# B&R Automation Studio project DuctLines (part 10)

### Program Logical/E2Buttons (IEC) - This program translates the Coil Line Run, Coil Line Halt And Coil Line Reset Buttons from the touch screen buttons for E2000s.

#### Cyclic.ld
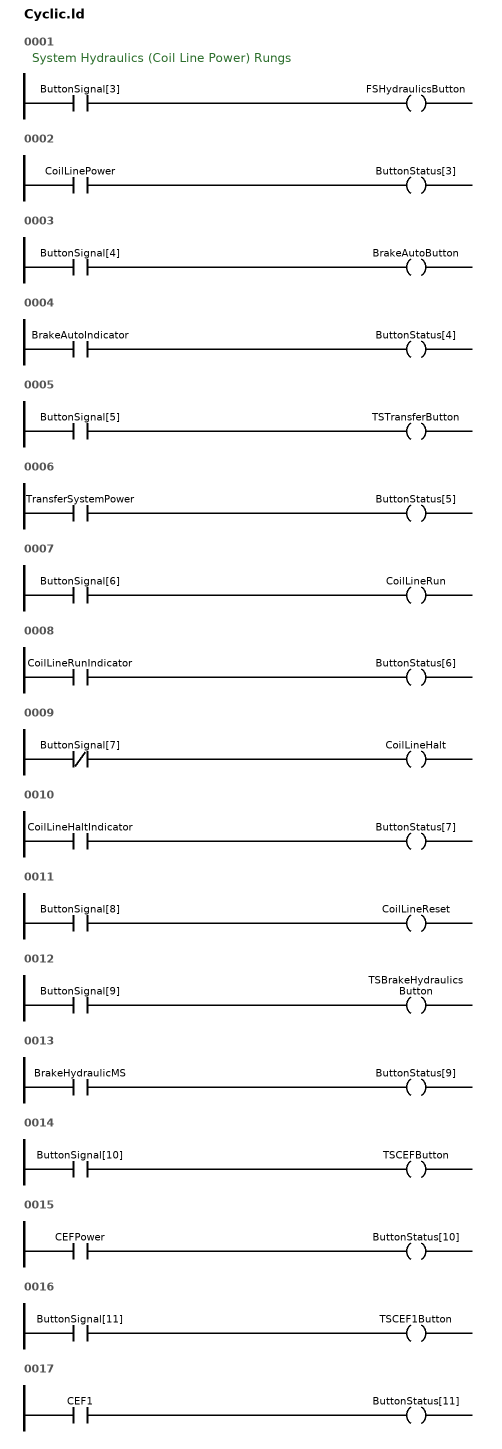
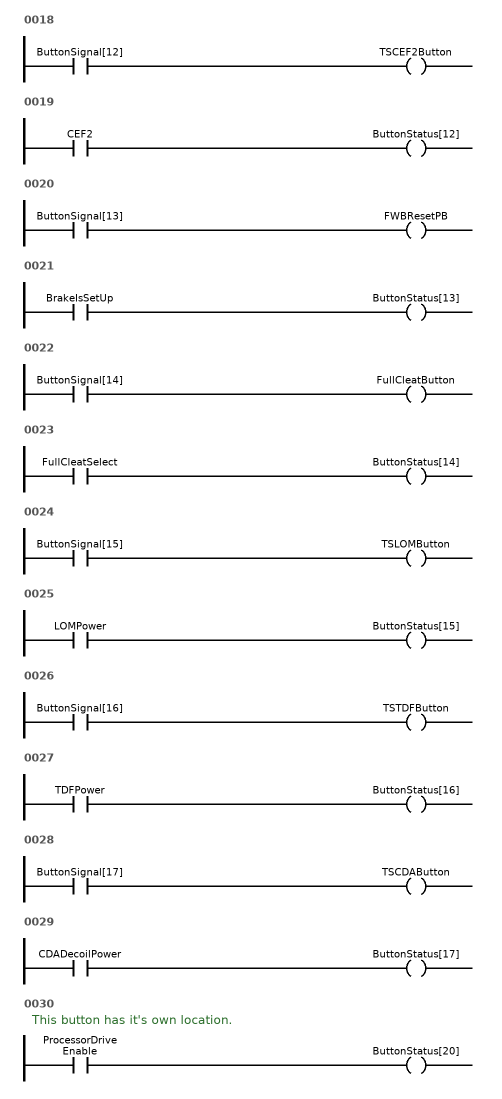
Ladder, written as Structured Text:
```iecst
PROGRAM _CYCLIC
(* Network 1: System Hydraulics (Coil Line Power) Rungs *)
FSHydraulicsButton := ButtonSignal[3];

(* Network 2 *)
ButtonStatus[3] := CoilLinePower;

(* Network 3 *)
BrakeAutoButton := ButtonSignal[4];

(* Network 4 *)
ButtonStatus[4] := BrakeAutoIndicator;

(* Network 5 *)
TSTransferButton := ButtonSignal[5];

(* Network 6 *)
ButtonStatus[5] := TransferSystemPower;

(* Network 7 *)
CoilLineRun := ButtonSignal[6];

(* Network 8 *)
ButtonStatus[6] := CoilLineRunIndicator;

(* Network 9 *)
CoilLineHalt := NOT ButtonSignal[7];

(* Network 10 *)
ButtonStatus[7] := CoilLineHaltIndicator;

(* Network 11 *)
CoilLineReset := ButtonSignal[8];

(* Network 12 *)
TSBrakeHydraulicsButton := ButtonSignal[9];

(* Network 13 *)
ButtonStatus[9] := BrakeHydraulicMS;

(* Network 14 *)
TSCEFButton := ButtonSignal[10];

(* Network 15 *)
ButtonStatus[10] := CEFPower;

(* Network 16 *)
TSCEF1Button := ButtonSignal[11];

(* Network 17 *)
ButtonStatus[11] := CEF1;

(* Network 18 *)
TSCEF2Button := ButtonSignal[12];

(* Network 19 *)
ButtonStatus[12] := CEF2;

(* Network 20 *)
FWBResetPB := ButtonSignal[13];

(* Network 21 *)
ButtonStatus[13] := BrakeIsSetUp;

(* Network 22 *)
FullCleatButton := ButtonSignal[14];

(* Network 23 *)
ButtonStatus[14] := FullCleatSelect;

(* Network 24 *)
TSLOMButton := ButtonSignal[15];

(* Network 25 *)
ButtonStatus[15] := LOMPower;

(* Network 26 *)
TSTDFButton := ButtonSignal[16];

(* Network 27 *)
ButtonStatus[16] := TDFPower;

(* Network 28 *)
TSCDAButton := ButtonSignal[17];

(* Network 29 *)
ButtonStatus[17] := CDADecoilPower;

(* Network 30: This button has it's own location. *)
ButtonStatus[20] := ProcessorDriveEnable;
END_PROGRAM
```

### Program Logical/EFdrSrvDrv (IEC) - Rungs To Control The Electric Servo Drive Option For The Feed Rolls

#### Variables.var
```iecst
VAR
	RollEnableUnlatch : BOOL;
END_VAR
```

#### Cyclic.ld
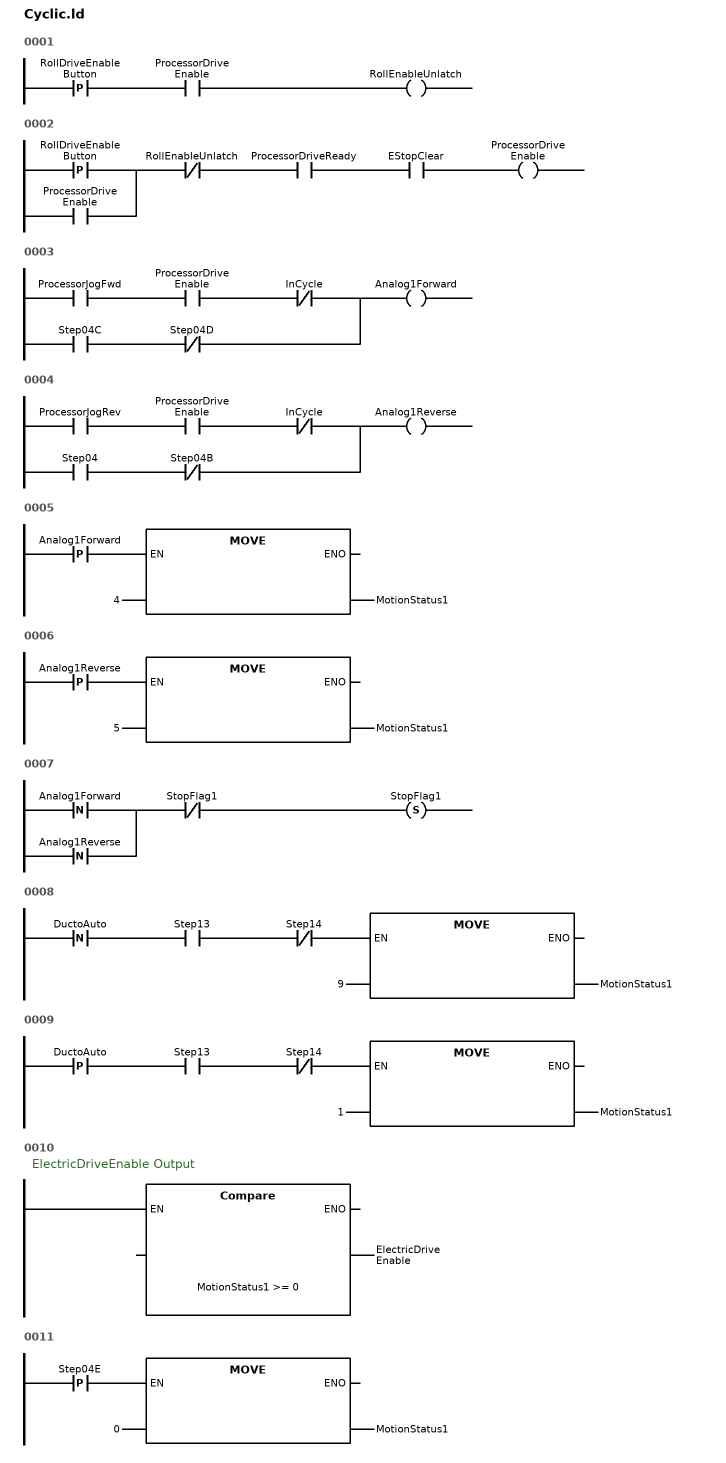
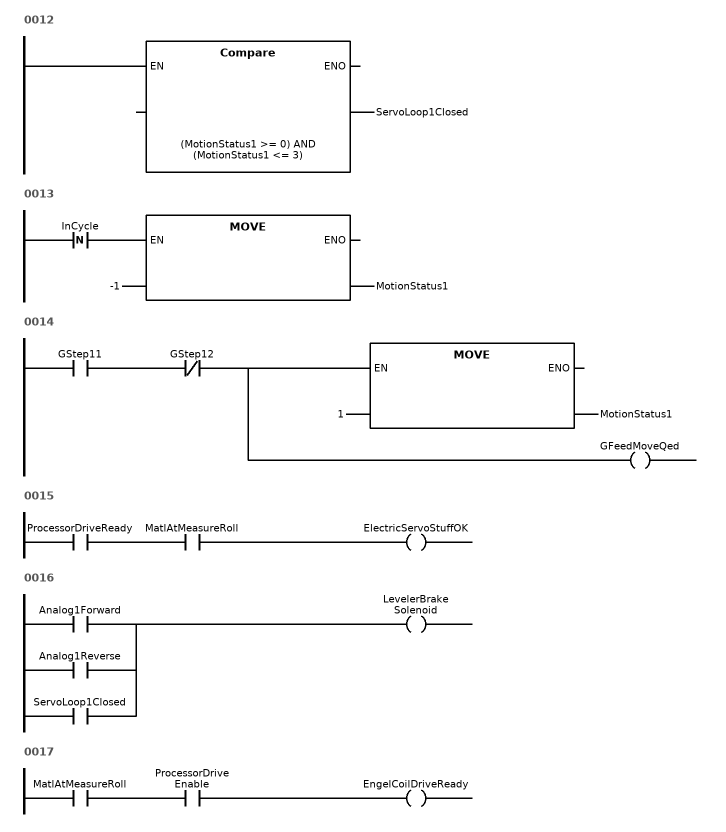
Ladder, written as Structured Text:
```iecst
PROGRAM _CYCLIC
VAR
    _e1 : R_TRIG;
    _e2 : R_TRIG;
    _e3 : R_TRIG;
    _e4 : R_TRIG;
    _e5 : F_TRIG;
    _e6 : F_TRIG;
    _e7 : F_TRIG;
    _e8 : R_TRIG;
    _e9 : R_TRIG;
    _e10 : F_TRIG;
END_VAR
(* Network 1 *)
_e1(CLK := RollDriveEnableButton);
RollEnableUnlatch := _e1.Q AND ProcessorDriveEnable;

(* Network 2 *)
_e2(CLK := RollDriveEnableButton);
ProcessorDriveEnable := (_e2.Q OR ProcessorDriveEnable) AND NOT RollEnableUnlatch AND ProcessorDriveReady AND EStopClear;

(* Network 3 *)
Analog1Forward := (ProcessorJogFwd AND ProcessorDriveEnable AND NOT InCycle) OR (Step04C AND NOT Step04D);

(* Network 4 *)
Analog1Reverse := (ProcessorJogRev AND ProcessorDriveEnable AND NOT InCycle) OR (Step04 AND NOT Step04B);

(* Network 5 *)
_e3(CLK := Analog1Forward);
IF _e3.Q THEN MotionStatus1 := 4; END_IF;

(* Network 6 *)
_e4(CLK := Analog1Reverse);
IF _e4.Q THEN MotionStatus1 := 5; END_IF;

(* Network 7 *)
_e5(CLK := Analog1Forward);
_e6(CLK := Analog1Reverse);
IF (_e5.Q OR _e6.Q) AND NOT StopFlag1 THEN StopFlag1 := TRUE; END_IF;

(* Network 8 *)
_e7(CLK := DuctoAuto);
IF _e7.Q AND Step13 AND NOT Step14 THEN MotionStatus1 := 9; END_IF;

(* Network 9 *)
_e8(CLK := DuctoAuto);
IF _e8.Q AND Step13 AND NOT Step14 THEN MotionStatus1 := 1; END_IF;

(* Network 10: ElectricDriveEnable Output *)
ElectricDriveEnable := MotionStatus1 >= 0;

(* Network 11 *)
_e9(CLK := Step04E);
IF _e9.Q THEN MotionStatus1 := 0; END_IF;

(* Network 12 *)
ServoLoop1Closed := (MotionStatus1 >= 0) AND (MotionStatus1 <= 3);

(* Network 13 *)
_e10(CLK := InCycle);
IF _e10.Q THEN MotionStatus1 := -1; END_IF;

(* Network 14 *)
IF GStep11 AND NOT GStep12 THEN MotionStatus1 := 1; END_IF;
GFeedMoveQed := GStep11 AND NOT GStep12;

(* Network 15 *)
ElectricServoStuffOK := ProcessorDriveReady AND MatlAtMeasureRoll;

(* Network 16 *)
LevelerBrakeSolenoid := Analog1Forward OR Analog1Reverse OR ServoLoop1Closed;

(* Network 17 *)
EngelCoilDriveReady := MatlAtMeasureRoll AND ProcessorDriveEnable;
END_PROGRAM
```

### Program Logical/EFdrHydDrv (IEC) - Rungs to control an Engel processor with the original two speed hydraulic solenoids.

#### Variables.var
```iecst
VAR
	difference : DINT;
	AbsoluteDifference : DINT;
	InTargetWindow : BOOL;
	TON_0 : TON;
	MovingToPosition : BOOL;
	MoveInitiated : BOOL;
	PositionLTTarget : BOOL;
	MoveForward : BOOL;
	PositionGTTarget : BOOL;
	MoveReverse : BOOL;
	InSSWindow : BOOL;
	SettleTimerDone : BOOL;
	TON_1 : TON;
	RevDelay : BOOL;
	TON_2 : TON;
	FwdDelay : BOOL;
	TON_3 : TON;
	SSSDelay : BOOL;
	TON_4 : TON;
	EnableForwardSolenoid : BOOL;
	TP_0 : TP;
	ForwardTP : BOOL;
	TON_5 : TON;
	EnableReverseSolenoid : BOOL;
END_VAR
```

#### Cyclic.ld
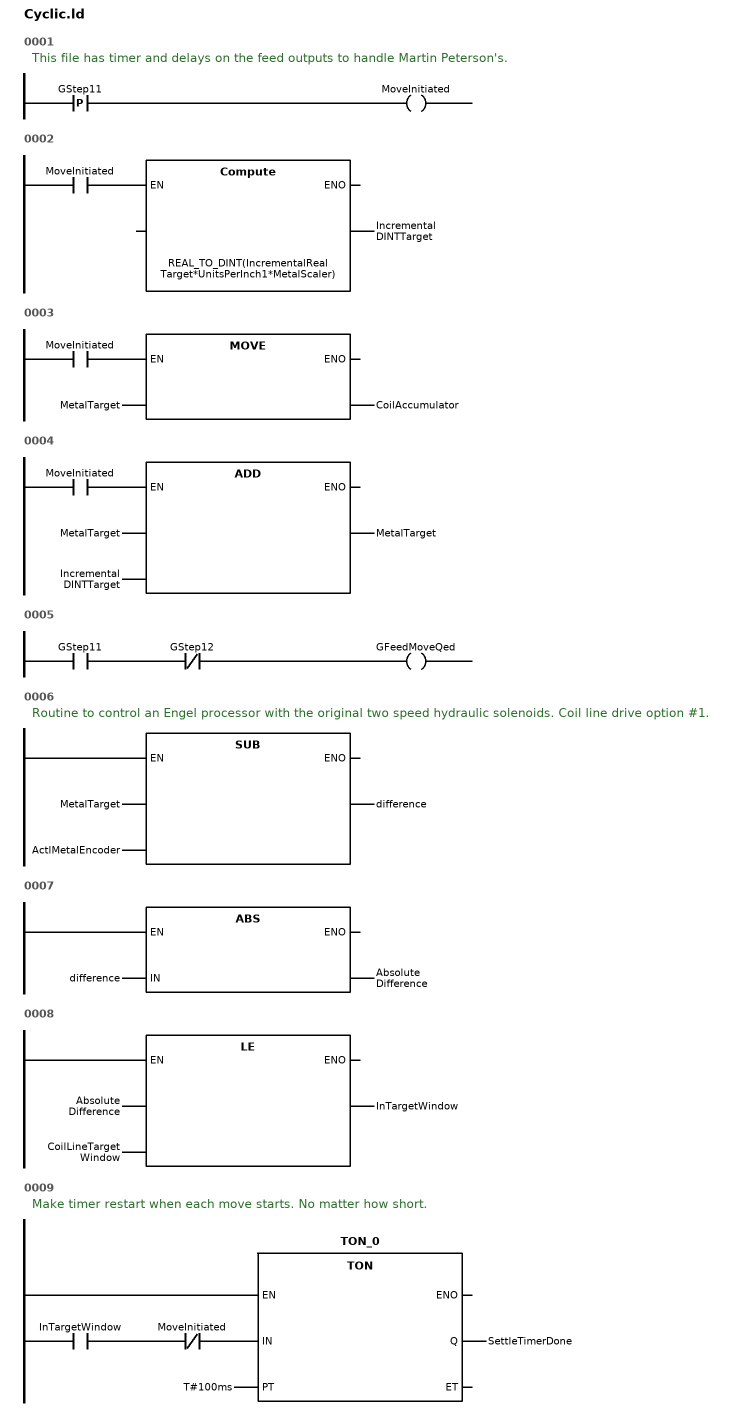
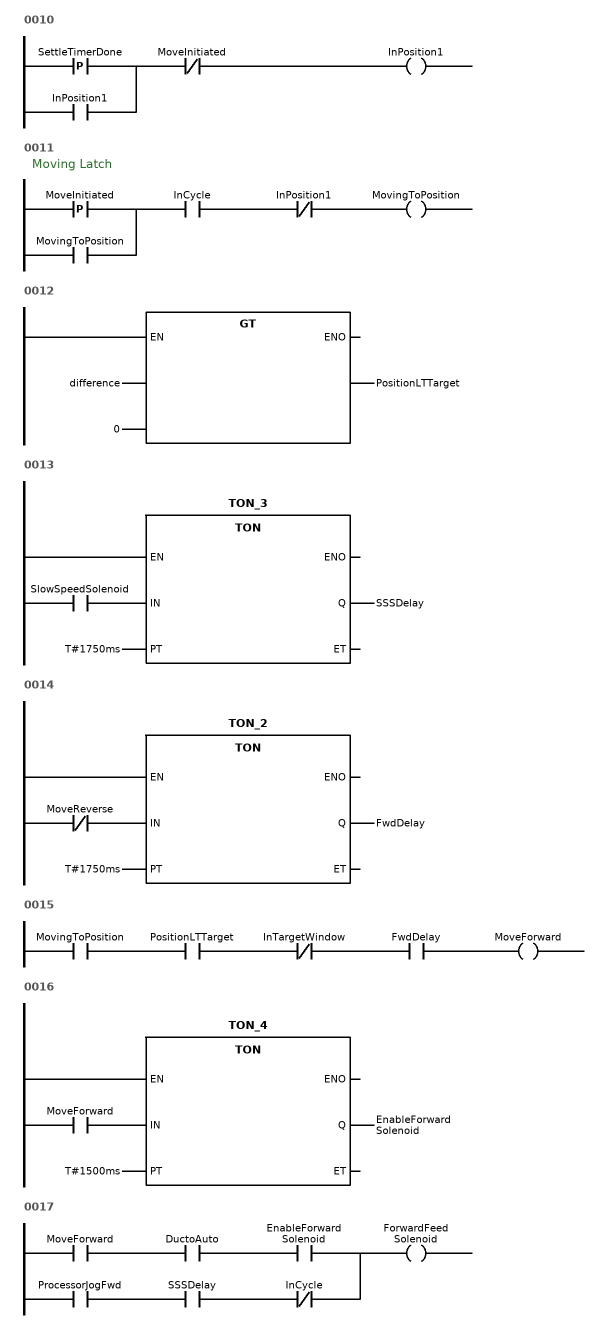
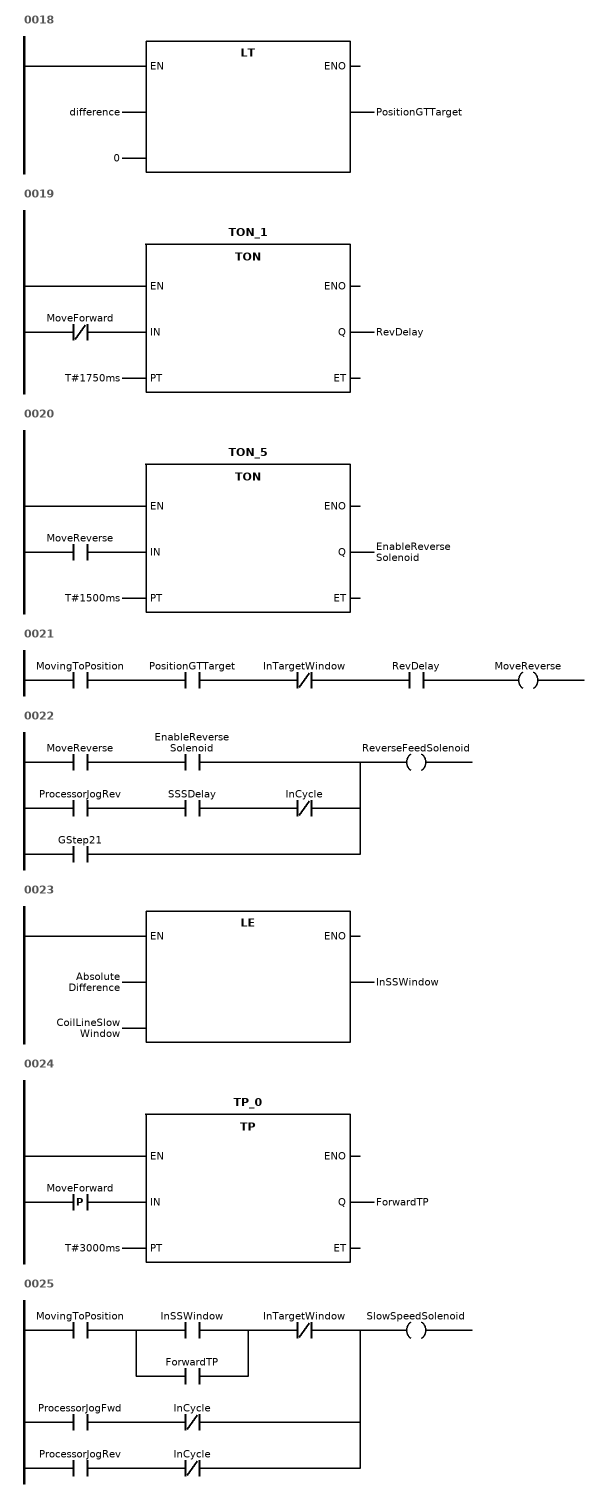
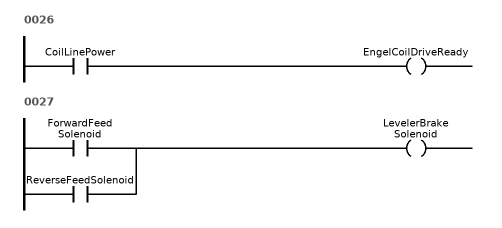
Ladder, written as Structured Text:
```iecst
PROGRAM _CYCLIC
VAR
    _e1 : R_TRIG;
    _e2 : R_TRIG;
    _e3 : R_TRIG;
    _e4 : R_TRIG;
END_VAR
(* Network 1: This file has timer and delays on the feed outputs to handle Martin Peterson's. *)
_e1(CLK := GStep11);
MoveInitiated := _e1.Q;

(* Network 2 *)
IF MoveInitiated THEN
    IncrementalDINTTarget := REAL_TO_DINT(IncrementalRealTarget*UnitsPerInch1*MetalScaler);
END_IF;

(* Network 3 *)
IF MoveInitiated THEN CoilAccumulator := MetalTarget; END_IF;

(* Network 4 *)
IF MoveInitiated THEN MetalTarget := MetalTarget + IncrementalDINTTarget; END_IF;

(* Network 5 *)
GFeedMoveQed := GStep11 AND NOT GStep12;

(* Network 6: Routine to control an Engel processor with the original two speed hydraulic solenoids. Coil line drive option #1. *)
difference := MetalTarget - ActlMetalEncoder;

(* Network 7 *)
AbsoluteDifference := ABS(difference);

(* Network 8 *)
InTargetWindow := AbsoluteDifference <= CoilLineTargetWindow;

(* Network 9: Make timer restart when each move starts. No matter how short. *)
TON_0(IN := InTargetWindow AND NOT MoveInitiated, PT := T#100ms);
SettleTimerDone := TON_0.Q;

(* Network 10 *)
_e2(CLK := SettleTimerDone);
InPosition1 := (_e2.Q OR InPosition1) AND NOT MoveInitiated;

(* Network 11: Moving Latch *)
_e3(CLK := MoveInitiated);
MovingToPosition := (_e3.Q OR MovingToPosition) AND InCycle AND NOT InPosition1;

(* Network 12 *)
PositionLTTarget := difference > 0;

(* Network 13 *)
TON_3(IN := SlowSpeedSolenoid, PT := T#1750ms);
SSSDelay := TON_3.Q;

(* Network 14 *)
TON_2(IN := NOT MoveReverse, PT := T#1750ms);
FwdDelay := TON_2.Q;

(* Network 15 *)
MoveForward := MovingToPosition AND PositionLTTarget AND NOT InTargetWindow AND FwdDelay;

(* Network 16 *)
TON_4(IN := MoveForward, PT := T#1500ms);
EnableForwardSolenoid := TON_4.Q;

(* Network 17 *)
ForwardFeedSolenoid := (MoveForward AND DuctoAuto AND EnableForwardSolenoid) OR (ProcessorJogFwd AND SSSDelay AND NOT InCycle);

(* Network 18 *)
PositionGTTarget := difference < 0;

(* Network 19 *)
TON_1(IN := NOT MoveForward, PT := T#1750ms);
RevDelay := TON_1.Q;

(* Network 20 *)
TON_5(IN := MoveReverse, PT := T#1500ms);
EnableReverseSolenoid := TON_5.Q;

(* Network 21 *)
MoveReverse := MovingToPosition AND PositionGTTarget AND NOT InTargetWindow AND RevDelay;

(* Network 22 *)
ReverseFeedSolenoid := (MoveReverse AND EnableReverseSolenoid) OR (ProcessorJogRev AND SSSDelay AND NOT InCycle) OR GStep21;

(* Network 23 *)
InSSWindow := AbsoluteDifference <= CoilLineSlowWindow;

(* Network 24 *)
_e4(CLK := MoveForward);
TP_0(IN := _e4.Q, PT := T#3000ms);
ForwardTP := TP_0.Q;

(* Network 25 *)
SlowSpeedSolenoid := (MovingToPosition AND (InSSWindow OR ForwardTP) AND NOT InTargetWindow) OR (ProcessorJogFwd AND NOT InCycle) OR (ProcessorJogRev AND NOT InCycle);

(* Network 26 *)
EngelCoilDriveReady := CoilLinePower;

(* Network 27 *)
LevelerBrakeSolenoid := ForwardFeedSolenoid OR ReverseFeedSolenoid;
END_PROGRAM
```

### Program Logical/E2Transfer (IEC) - Controls the E2000 Transfer System

#### Variables.var
```iecst
VAR
	TSPUnlatch : BOOL;
	TSSystemTripPulse : BOOL;
	TP_0 : TP;
	TP_1 : TP;
	TP_2 : TP;
	Lift3DownPulse : BOOL;
	TON_0 : TON;
END_VAR
```

#### Cyclic.ld
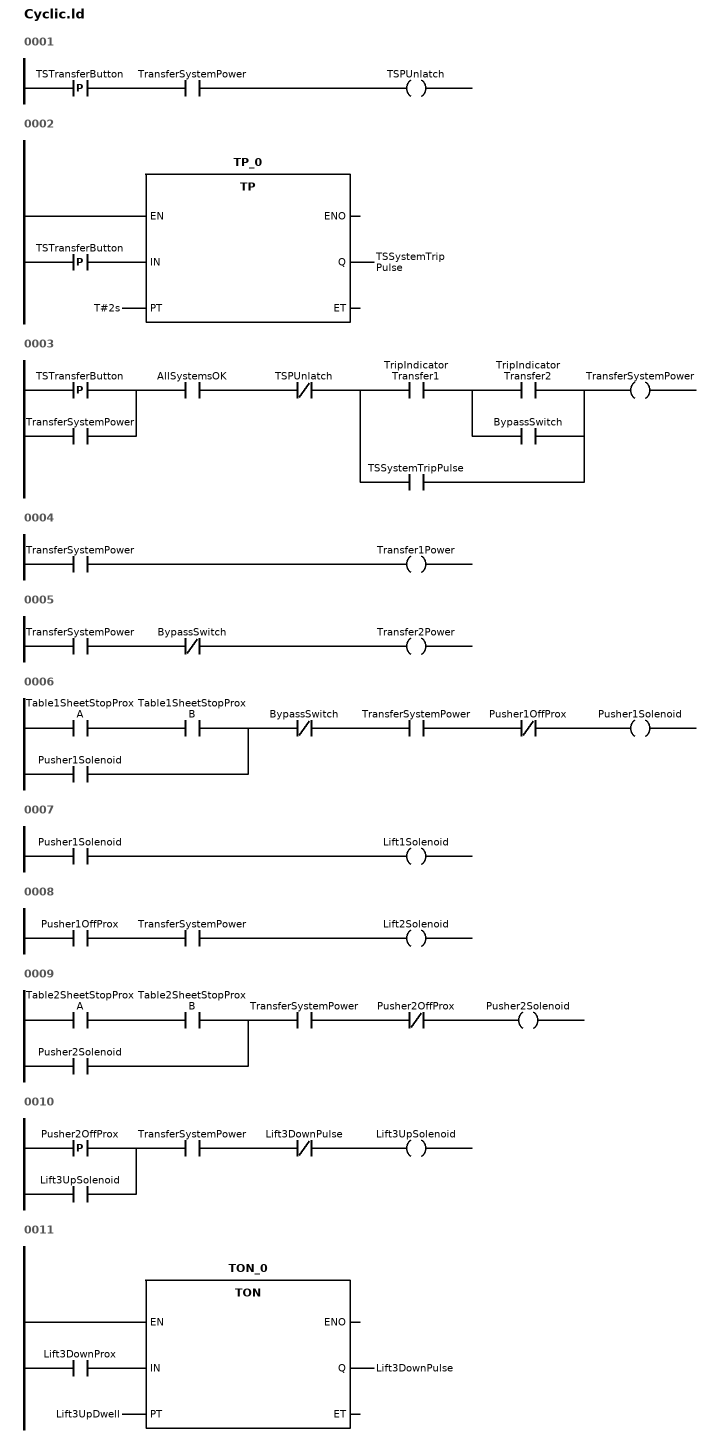
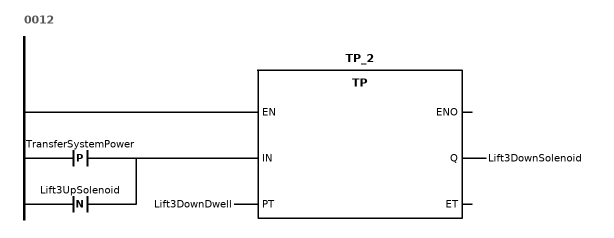
Ladder, written as Structured Text:
```iecst
PROGRAM _CYCLIC
VAR
    _e1 : R_TRIG;
    _e2 : R_TRIG;
    _e3 : R_TRIG;
    _p4 : BOOL;
    _e5 : R_TRIG;
    _e6 : R_TRIG;
    _e7 : F_TRIG;
END_VAR
(* Network 1 *)
_e1(CLK := TSTransferButton);
TSPUnlatch := _e1.Q AND TransferSystemPower;

(* Network 2 *)
_e2(CLK := TSTransferButton);
TP_0(IN := _e2.Q, PT := T#2s);
TSSystemTripPulse := TP_0.Q;

(* Network 3 *)
_e3(CLK := TSTransferButton);
_p4 := (_e3.Q OR TransferSystemPower) AND AllSystemsOK AND NOT TSPUnlatch;
TransferSystemPower := _p4 AND ((TripIndicatorTransfer1 AND (TripIndicatorTransfer2 OR BypassSwitch)) OR TSSystemTripPulse);

(* Network 4 *)
Transfer1Power := TransferSystemPower;

(* Network 5 *)
Transfer2Power := TransferSystemPower AND NOT BypassSwitch;

(* Network 6 *)
Pusher1Solenoid := ((Table1SheetStopProxA AND Table1SheetStopProxB) OR Pusher1Solenoid) AND NOT BypassSwitch AND TransferSystemPower AND NOT Pusher1OffProx;

(* Network 7 *)
Lift1Solenoid := Pusher1Solenoid;

(* Network 8 *)
Lift2Solenoid := Pusher1OffProx AND TransferSystemPower;

(* Network 9 *)
Pusher2Solenoid := ((Table2SheetStopProxA AND Table2SheetStopProxB) OR Pusher2Solenoid) AND TransferSystemPower AND NOT Pusher2OffProx;

(* Network 10 *)
_e5(CLK := Pusher2OffProx);
Lift3UpSolenoid := (_e5.Q OR Lift3UpSolenoid) AND TransferSystemPower AND NOT Lift3DownPulse;

(* Network 11 *)
TON_0(IN := Lift3DownProx, PT := Lift3UpDwell);
Lift3DownPulse := TON_0.Q;

(* Network 12 *)
_e6(CLK := TransferSystemPower);
_e7(CLK := Lift3UpSolenoid);
TP_2(IN := _e6.Q OR _e7.Q, PT := Lift3DownDwell);
Lift3DownSolenoid := TP_2.Q;
END_PROGRAM
```

### Program Logical/EMotionControl (IEC)

#### Variables.var
```iecst
VAR
	AbsoluteDifference : DINT;
	Counter1 : INT;
	DACBalance1 : INT;
	difference : DINT;
	Hold1 : INT;
	Ratio1 : INT;
END_VAR
```

#### Cyclic.st
```iecst
PROGRAM _CYCLIC
	difference := MetalTarget - ActlMetalEncoder;
	AbsoluteDifference := ABS(difference);
	CASE MotionStatus1 OF
		(*Hold Position*)
		0:
			IF NOT InPosition1 THEN
				IF AbsoluteDifference <= MetalTolerance THEN
					TargetCount1 := TargetCount1 + UpdateRate1;
					IF TargetCount1 >= SettleTime1 THEN
						InPosition1 := TRUE;
					END_IF;
				END_IF;
			END_IF;

			(*Ratio1 := DINT_TO_INT(difference + (difference / 1));*)
			Ratio1 := DINT_TO_INT(difference * 15);
			IF Counter1 > 0 THEN
				Counter1 := Counter1 - UpdateRate1;
			ELSE
				Counter1 := 500;
				IF Hold1 <> Ratio1 THEN
					Hold1 := Ratio1;
				ELSE
					DACBalance1 := ActualDAC1;
				END_IF;
			END_IF;

	    	TargetDAC1 := Ratio1 + DACBalance1;
			ActualDAC1 := TargetDAC1;
		(*	IF TargetDAC1 >= ActualDAC1 THEN
				IF TargetDAC1 - ActualDAC1 > (10 * UpdateRate1) THEN
					ActualDAC1 := ActualDAC1 + (10 * UpdateRate1);
				ELSE
					ActualDAC1 := TargetDAC1;
				END_IF;
			ELSE
				IF ActualDAC1 - TargetDAC1 > (10 * UpdateRate1) THEN
					ActualDAC1 := ActualDAC1 - (10 * UpdateRate1);
				ELSE
					ActualDAC1 := TargetDAC1;
				END_IF;
			END_IF;*)

			IF ActualDAC1 > TopDAC1 THEN
				ActualDAC1 := TopDAC1;
			END_IF;
			IF ActualDAC1 < -TopDAC1 THEN
				ActualDAC1 := -TopDAC1;
			END_IF

		(*Initialize Move*)
		1:
			CoilAccumulator := MetalTarget; (*Update Accumulator to last target*)
			(*IncrementalRealTarget is the amount required to move determined elsewhere*)
			IncrementalDINTTarget := REAL_TO_DINT(IncrementalRealTarget * UnitsPerInch1 * MetalScaler);
			MetalTarget := MetalTarget + IncrementalDINTTarget;
			DACAdd1 := INT_TO_REAL(MaxDAC) / AccelRampReal;
			TopDAC1 := DINT_TO_INT((INT_TO_DINT(MaxDAC) * RunSpeed1) / 100);
			IF RunSpeed1 = 100 THEN
				TopDAC1 := TopDAC1 - REAL_TO_INT(DACAdd1);
			END_IF;
			ActualSpeed1 := ((MaxSpeed1 / 5.0) * DINT_TO_REAL(RunSpeed1)) / 100.0; (*Real Inches Per Second*)
			AverageSpeed1 := ActualSpeed1 / 2.0;
			DecelTime1 := (DecelRampReal / 1000.0) * (DINT_TO_REAL(RunSpeed1) / 100);
			DecelDistance1 := REAL_TO_DINT(((AverageSpeed1 * DecelTime1 ) * MetalScaler) * UnitsPerInch1);
			MaxCountsPerSecond := (MaxSpeed1 / 5.0) * UnitsPerInch1;
			SRM1 := MaxDACSquared / ((MaxCountsPerSecond * (DecelRampReal / 1000.0)) / 2.0);
			(*SRM1 := MaxDACSquared / ((MaxCountsPerSecond * (DecelRampReal / 1000.0)));*)
			(*IF DecelDistance1 > IncrementalDINTTarget THEN 2-26-19 *)
			IF DecelDistance1 > (IncrementalDINTTarget / 2) THEN
				DecelDistance1 := IncrementalDINTTarget / 2;
				TopDAC1 := REAL_TO_INT(SQRT((DINT_TO_REAL(DecelDistance1) / MetalScaler) * SRM1));
				IF TopDAC1 < 3276 THEN
					TopDAC1 := 3276;
				END_IF;
			END_IF;
			InPosition1 := FALSE;
			FirstTarget1 := FALSE;
			StopWatch1 := 0.0;
			MotionStatus1 := 2;
		(*Ramp Up To Speed*)
		2:
			IF DecelDistance1 < difference THEN
				IF ActualDAC1 < TopDAC1 THEN (*Accelerate*)
					StopWatch1 := StopWatch1 + INT_TO_REAL(UpdateRate1);
					ActualDAC1 := REAL_TO_INT(StopWatch1 * DACAdd1);
				ELSE  (*Constant Speed*)
					ActualDAC1 := TopDAC1;
				END_IF;
			ELSE (*Switch To Decel MotionState*)
				DecelCounter := 25;
				LastPosition1 := ActlMetalEncoder;
				TargetCount1 := 0;
				FirstTarget1 := FALSE;
				MotionStatus1 := 3;
			END_IF;
		3:
			(*Stall Detection*)
			DecelCounter := DecelCounter - UpdateRate1;
			IF DecelCounter <= 0 THEN
				DecelCounter := 200;
				IF LastPosition1 = ActlMetalEncoder THEN
					DACBalance1 := ActualDAC1;
					Counter1 := 0;
					TopDAC1 := MaxDAC / 4;
					MotionStatus1 := 0;
				ELSE
					LastPosition1 := ActlMetalEncoder;
				END_IF;
			END_IF;

			RealDAC1 := REAL_TO_INT(SQRT(DINT_TO_REAL(AbsoluteDifference) * SRM1));
			IF RealDAC1 > INT_TO_REAL(MaxDAC) THEN
				RealDAC1 := INT_TO_REAL(MaxDAC);
			END_IF;
			ActualDAC1 := REAL_TO_INT(RealDAC1);

			IF difference < 0 THEN
				ActualDAC1 := -ActualDAC1;
			END_IF;

			IF FirstTarget1 THEN
				ActualDAC1 := ActualDAC1 / 8;
			END_IF;

			IF AbsoluteDifference < MetalTolerance THEN
				FirstTarget1 := TRUE;
				TargetCount1 := TargetCount1 + UpdateRate1;
				IF TargetCount1 >= SettleTime1 THEN
					Counter1 := 0;
					InPosition1 := TRUE;
					MotionStatus1 := 0;
					TopDAC1 := MaxDAC / 4;
				END_IF;
			ELSE
				TargetCount1 := 0;
			END_IF;
		4: (*Setup Forward Jog*)
			DACAdd1 := INT_TO_REAL(MaxDAC) / AccelRampReal;
			TopDAC1 := DINT_TO_INT((INT_TO_DINT(MaxDAC) * PercentJogSpeed1) / 100);
			TopDAC1 := TopDAC1 - REAL_TO_INT(DACAdd1);
			StopFlag1 := FALSE;
			MotionStatus1 := 7;
		5: (*Setup Reverse Jog*)
			DACAdd1 := INT_TO_REAL(MaxDAC) / AccelRampReal;
			TopDAC1 := DINT_TO_INT((INT_TO_DINT(MaxDAC) * PercentJogSpeed1) / 100);
			TopDAC1 := TopDAC1 - REAL_TO_INT(DACAdd1);
			StopFlag1 := FALSE;
			MotionStatus1 := 8;
		7: (*Forward Jog*)
			IF StopFlag1 THEN
				IF ActualDAC1 > REAL_TO_INT(DACAdd1) THEN (*Decelerate*)
					ActualDAC1 := ActualDAC1 - REAL_TO_INT(DACAdd1);
				ELSE (*Hold Position*)
					ActualDAC1 := 0;
					MetalTarget := ActlMetalEncoder;
					InPosition1 := TRUE;
					MotionStatus1 := -1;
				END_IF;
			ELSE
				InPosition1 := FALSE;
				IF ActualDAC1 < TopDAC1 THEN (*Accelerate*)
					ActualDAC1 := ActualDAC1 + REAL_TO_INT(DACAdd1);
				ELSE
					ActualDAC1 := TopDAC1; (*Maintain Constant Speed*)
				END_IF;
			END_IF;
		8: (*Reverse Jog*)
			IF StopFlag1 THEN
				IF ActualDAC1 < REAL_TO_INT(-DACAdd1) THEN (*Decelerate*)
					ActualDAC1 := ActualDAC1 + REAL_TO_INT(DACAdd1);
				ELSE (*Hold Position*)
					ActualDAC1 := 0;
					MetalTarget := ActlMetalEncoder;
					InPosition1 := TRUE;
					MotionStatus1 := -1;
				END_IF;
			ELSE
				(*Don't Do This To Prevent Uncoiler From Running Forward*)
				(*InPosition1 := FALSE;*)
				IF ActualDAC1 > -TopDAC1 THEN (*Accelerate*)
					ActualDAC1 := ActualDAC1 - REAL_TO_INT(DACAdd1);
				ELSE
					ActualDAC1 := -TopDAC1; (*Maintain Constant Speed*)
				END_IF;
			END_IF;
		9:
			IF ActualDAC1 > REAL_TO_INT(DACAdd1) THEN (*Decelerate*)
				ActualDAC1 := ActualDAC1 - REAL_TO_INT(DACAdd1);
			ELSE (* Hold Position *)
				MetalTarget := ActlMetalEncoder;
				IncrementalRealTarget := DINT_TO_REAL(difference) / UnitsPerInch1 / MetalScaler;
				MotionStatus1 := 0;
			END_IF;
		ELSE (*Not Moving Or Holding*)
		  ActualDAC1 := 0;
		  MetalTarget := ActlMetalEncoder;
		  InPosition1 := TRUE;
	END_CASE;

	IF ActualDAC1 > MaxDAC THEN
		ActualDAC1 := MaxDAC;
	END_IF;
	IF ActualDAC1 < -MaxDAC THEN
		ActualDAC1 := -MaxDAC;
	END_IF;

END_PROGRAM
```

#### Init.st
```iecst
PROGRAM _INIT
	MotionStatus1 := -1;
	InPosition1 := TRUE;
END_PROGRAM
```

### Program Logical/Feeder1 (IEC)

#### Variables.var
```iecst
VAR
	AnalogForward : BOOL;
	AnalogReverse : BOOL;
	AutoSignal : BOOL;
	BatchCancelUnlatch : BOOL;
	BeadRollFires : BOOL;
	BeadRollUsedUp : BOOL;
	Block_1 : BOOL;
	BrakeLatch : BOOL;
	ButtonBack7 : BOOL;
	ButtonFires : BOOL;
	ButtonUsedUp : BOOL;
	CenterHoleFires : BOOL;
	CenterHoleTime : TIME;
	CenterHoleUsedUp : BOOL;
	CenterPosA : BOOL;
	CenterShuttleIndex : INT;
	ChangeCShuttle : BOOL;
	ChangeJob1 : BOOL;
	ChangeRShuttle : BOOL;
	CHTemp : BOOL;
	ClearEncoderSignal : BOOL;
	CleatFires : BOOL;
	CleatUsedUp : BOOL;
	CLTTemp : BOOL;
	CShuttleUnlatch : BOOL;
	CustomLTFires : BOOL;
	CustomLTTime : TIME;
	CustomLTUsedUp : BOOL;
	CustomLTValve : BOOL;
	CustomVFires : BOOL;
	CustomVTemp : BOOL;
	CustomVTime : TIME;
	CustomVUsedUp : BOOL;
	DataUpdated : BOOL;
	DDDoneTimer : TON;
	DieDelayDone : BOOL;
	DieUpTime : TIME;
	DirectionDelayDone : BOOL;
	FeedMoveQed : BOOL;
	FinalScan : BOOL;
	GapPulse : BOOL;
	GapTP : BOOL;
	GTime : TIME;
	HalfUpdated1 : BOOL;
	HalfUpdated2 : BOOL;
	IncPartsMade : BOOL;
	InitMoveSignal : BOOL;
	InPositionBand : REAL := 0.01;
	JobChanging : BOOL;
	JobsDifferent : BOOL;
	LeftHoleFires : BOOL;
	LeftHoleTime : TIME;
	LeftHoleUsedUp : BOOL;
	LeftPosA : BOOL;
	LHTemp : BOOL;
	LTFires : BOOL;
	LTTemp : BOOL;
	LTTime : TIME;
	LTUsedUp : BOOL;
	MarkAccumulator : REAL;
	MetalEncoderLatch : DINT;
	NewRunJobOk : BOOL;
	NextMoveComplete : BOOL;
	NextMoveLookAgain : BOOL;
	NoShearHits : BOOL;
	PartCutOff : BOOL;
	PulseProcessorReset : BOOL;
	ReturnCalculated : BOOL;
	ReturnComplete : BOOL;
	ReturnTarget : DINT;
	RHTemp : BOOL;
	RightHoleFires : BOOL;
	RightHoleTime : TIME;
	RightHoleUsedUp : BOOL;
	RightPosA : BOOL;
	RShuttleUnlatch : BOOL;
	RTotalInches : REAL;
	RunSpeedCalculated : BOOL;
	SBClampDelay : TIME;
	SBClampDwell : TIME;
	SetConnectorChange : BOOL;
	ShearBrakeFires : BOOL;
	ShearBrakeUsedUp : BOOL;
	ShearFires : BOOL;
	ShearHitsLTZero : BOOL;
	ShearTemp : BOOL;
	shearTime : TIME;
	ShearUsedUp : BOOL;
	SHLT0 : BOOL;
	SmallResult : REAL;
	Step04A : BOOL;
	Step05A : BOOL;
	Step05B : BOOL;
	Step06 : BOOL;
	Step07 : BOOL;
	Step08 : BOOL;
	Step09 : BOOL;
	Step10 : BOOL;
	Step11 : BOOL;
	Step15 : BOOL;
	Step16 : BOOL;
	Step17 : BOOL;
	Step18A : BOOL;
	Step20 : BOOL;
	Step22 : BOOL;
	ThirdOff1 : BOOL;
	ThirdOff2 : BOOL;
	ThirdOff3 : BOOL;
	TON_0 : TON;
	TON_1 : TON;
	TON_2 : TON;
	TON_10 : TON;
	TON_Warning : TON;
	TP_0 : TP;
	TP_1 : TP;
	TP_2 : TP;
	TP_3 : TP;
	TP_4 : TP;
	TP_5 : TP;
	TP_6 : TP;
	TP_7 : TP;
	TP_8 : TP;
	TP_9 : TP;
	UnlatchBender : BOOL;
	UnlatchButtons : BOOL;
	VFires : BOOL;
	VTemp : BOOL;
	VTime : TIME;
	VUsedUp : BOOL;
	Wait1Ready : BOOL;
	Wait2Ready : BOOL;
	Wait3Ready : BOOL;
	WaitCon1 : BOOL;
	WaitCon2 : BOOL;
	ZCOLT0 : BOOL;
	ZCReverseComplete : BOOL;
	ZCSCTimer : TON;
	ZCSettleComplete : BOOL;
	ZeroCropDifference : DINT;
	ZRCTon : TON;
END_VAR
```

#### Action.st
```iecst
ACTION myAction:
	(* This was for a test *)
	IF myAction.x AND NOT myAction._x THEN
		FinalScan := TRUE;
	ELSE
	    IF ShearHits < 120000 THEN
			ShearHits := ShearHits + 1;
		END_IF;
	END_IF;

END_ACTION

ACTION getNextMove:
	IF getNextMove.x AND NOT getNextMove._x THEN
		FinalScan := TRUE;
    ELSE
	(*Find smallest move*)
		(*The shear will always be used*)
		NextMoveDone := TRUE;
	SmallResult := ShearMove;
	IF LTNotchMove < SmallResult AND LTNotchMove > InvalidDistREAL THEN
		SmallResult := LTNotchMove;
	END_IF;
	IF VNotchMove < SmallResult AND VNotchMove > InvalidDistREAL THEN
		SmallResult := VNotchMove;
	END_IF;
	IF LeftHoleMove < SmallResult AND LeftHoleMove > InvalidDistREAL THEN
		SmallResult := LeftHoleMove;
	END_IF;
	IF CenterHoleMove < SmallResult AND CenterHoleMove > InvalidDistREAL THEN
		SmallResult := CenterHoleMove;
	END_IF;
	IF RightHoleMove < SmallResult AND RightHoleMove > InvalidDistREAL THEN
		SmallResult := RightHoleMove;
	END_IF;
	IF ButtonMove < SmallResult AND ButtonMove > InvalidDistREAL THEN
		SmallResult := ButtonMove;
	END_IF;
	IF ShearBrakeMove < SmallResult AND ShearBrakeMove > InvalidDistREAL THEN
		SmallResult := ShearBrakeMove;
	END_IF;
	IF CustomLTMove < SmallResult AND CustomLTMove > InvalidDistREAL THEN
		SmallResult := CustomLTMove;
	END_IF;
	IF CleatMove < SmallResult AND CleatMove > InvalidDistREAL THEN
		SmallResult := CleatMove;
	END_IF;
	IF CustomVMove < SmallResult AND CustomVMove > InvalidDistREAL THEN
		SmallResult := CustomVMove;
	END_IF;
	IF BeadRollMove < SmallResult AND BeadRollMove > InvalidDistREAL THEN
		SmallResult := BeadRollMove;
	END_IF;

	ShearMove := ShearMove - SmallResult;
	IF LTNotchMove > InvalidDistREAL THEN
		LTNotchMove := LTNotchMove - SmallResult;
	END_IF;
	IF VNotchMove > InvalidDistREAL THEN
		VNotchMove := VNotchMove - SmallResult;
	END_IF;
	IF LeftHoleMove > InvalidDistREAL THEN
		LeftHoleMove := LeftHoleMove - SmallResult;
	END_IF;
	IF CenterHoleMove > InvalidDistREAL THEN
		CenterHoleMove := CenterHoleMove - SmallResult;
	END_IF;
	IF RightHoleMove > InvalidDistREAL THEN
		RightHoleMove := RightHoleMove - SmallResult;
	END_IF;
	IF ButtonMove > InvalidDistREAL THEN
		ButtonMove := ButtonMove - SmallResult;
	END_IF;
	IF ShearBrakeMove > InvalidDistREAL THEN
		ShearBrakeMove := ShearBrakeMove - SmallResult;
	END_IF;
	IF CustomLTMove > InvalidDistREAL THEN
		CustomLTMove := CustomLTMove - SmallResult;
	END_IF;
	IF CleatMove > InvalidDistREAL THEN
		CleatMove := CleatMove - SmallResult;
	END_IF;
	IF CustomVMove > InvalidDistREAL THEN
		CustomVMove := CustomVMove - SmallResult;
	END_IF;
	IF BeadRollMove > InvalidDistREAL THEN
		BeadRollMove := BeadRollMove - SmallResult;
	END_IF;
  END_IF;
END_ACTION

ACTION UpdateTables:
	IF UpdateTables.x AND NOT UpdateTables._x THEN
		FinalScan := TRUE;
	ELSE
		UpdateTablesDone := TRUE;
		IF ShearUsedUp AND ShearHits > 0 THEN
			ShearFires := TRUE;
			ShearHits := ShearHits - 1;
			(*Do this before the index changes *)
			IF (ShearIndex = 0 AND ShearFFlag = 1) OR
				(ShearIndex = 1 AND ShearTable[2] <= InvalidDistREAL) OR
				(ShearIndex = 2) THEN
				PartCutOff := TRUE;
			END_IF;
				ShearIndex := ShearIndex + 1;
			IF ShearTable[ShearIndex] <= InvalidDistREAL THEN
				ShearIndex := 1;
			END_IF;
			IF ShearHits <= 0 THEN
				MakeShearTable := TRUE;
				ShearIndex := 0;
			END_IF;
		END_IF;
		IF LTUsedUp THEN
			IF LTNotchHits > 0 THEN
				LTFires := TRUE;
				LTNotchHits := LTNotchHits - 1;
			END_IF;
			LTNotchIndex := LTNotchIndex + 1;
			IF LTNotchTable[LTNotchIndex] <= InvalidDistREAL THEN
				LTNotchIndex := 1;
			END_IF;
			SavedConnector := LatestConnector;
			IF LTNotchHits <= 0 THEN
				MakeLTTable := TRUE;
				LTNotchIndex := 0;
			END_IF;
		END_IF;
		IF VUsedUp THEN
			IF VNotchHits > 0 THEN
				VFires := TRUE;
				VNotchHits := VNotchHits - 1;
			END_IF;
			VNotchIndex := VNotchIndex + 1;
			IF VNotchTable[VNotchIndex] <= InvalidDistREAL THEN
				VNotchIndex := 1;
			END_IF;
			IF VNotchHits <= 0 THEN
				MakeVTable := TRUE;
				VNotchIndex := 0;
			END_IF;
		END_IF;
		IF LeftHoleUsedUp THEN
			IF LeftHoleHits > 0 THEN
				LeftHoleFires := TRUE;
				LeftHoleHits := LeftHoleHits - 1;
			END_IF;
			LeftHoleIndex := LeftHoleIndex + 1;
			IF LeftHoleTable[LeftHoleIndex] <= InvalidDistREAL THEN
				LeftHoleIndex := 1;
			END_IF;
			IF LeftHoleHits <= 0 THEN
				MakeLHoleTable := TRUE;
				LeftHoleIndex := 0;
			END_IF;
		END_IF;
		IF CenterHoleUsedUp THEN
			IF CenterHoleHits > 0 THEN
				CenterHoleFires := TRUE;
				CenterHoleHits := CenterHoleHits - 1;
			END_IF;
			CenterHoleIndex := CenterHoleIndex + 1;
			IF CenterHoleTable[CenterHoleIndex] <= InvalidDistREAL THEN
				CenterHoleIndex := 1;
			END_IF;
			IF CenterHoleHits <= 0 THEN
				MakeCHoleTable := TRUE;
				CenterHoleIndex := 0;
			END_IF;
		END_IF;
		IF RightHoleUsedUp THEN
			IF RightHoleHits > 0 THEN
				RightHoleFires := TRUE;
				RightHoleHits := RightHoleHits - 1;
			END_IF;
			RightHoleIndex := RightHoleIndex + 1;
			IF RightHoleTable[RightHoleIndex] <= InvalidDistREAL THEN
				RightHoleIndex := 1;
			END_IF;
			IF RightHoleHits <= 0 THEN
				MakeRHoleTable := TRUE;
				RightHoleIndex := 0;
			END_IF;
		END_IF
		IF ButtonUsedUp THEN
			IF ButtonHits > 0 THEN
				ButtonFires := TRUE;
				ButtonHits := ButtonHits - 1;
			END_IF;
			ButtonIndex := ButtonIndex + 1;
			IF ButtonTable[ButtonIndex] <= InvalidDistREAL THEN
				ButtonIndex := 1;
			END_IF;
			IF ButtonHits <= 0 THEN
				MakeButtonTable := TRUE;
				ButtonIndex := 0;
			END_IF;
		END_IF;
		IF ShearBrakeUsedUp THEN
			IF ShearBrakeHits > 0 THEN
				ShearBrakeFires := TRUE;
				ShearBrakeHits := ShearBrakeHits - 1;
			END_IF;
			IF ShearBrakeTable[ShearBrakeIndex] <= InvalidDistREAL THEN
				ShearBrakeIndex := 1;
			END_IF;
			ShearBrakeIndex := ShearBrakeIndex + 1;
			IF ShearBrakeHits <= 0 THEN
				MakeShearBrakeTable := TRUE;
				ShearBrakeIndex := 0;
			END_IF;
		END_IF;
		IF CustomLTUsedUp THEN
			IF CustomLTHits > 0 THEN
				CustomLTFires := TRUE;
				CustomLTHits := CustomLTHits - 1;
			END_IF;
			CustomLTIndex := CustomLTIndex + 1;
			IF CustomLTTable[CustomLTIndex] <= InvalidDistREAL THEN
				CustomLTIndex := 1;
			END_IF;
			IF CustomLTHits <= 0 THEN
				MakeCustomLTTable := TRUE;
				CustomLTIndex := 0;
			END_IF;
		END_IF;
		IF CleatUsedUp THEN
			IF CleatHits > 0 THEN
				CleatFires := TRUE;
				CleatHits := CleatHits - 1;
			END_IF;
			CleatIndex := CleatIndex + 1;
			IF CleatTable[CleatIndex] <= InvalidDistREAL THEN
				CleatIndex := 1;
			END_IF;
			IF CleatHits <= 0 THEN
				MakeCleatTable := TRUE;
				CleatIndex := 0;
			END_IF;
		END_IF;
		IF CustomVUsedUp THEN
			IF CustomVHits > 0 THEN
				CustomVFires := TRUE;
				CustomVHits := CustomVHits - 1;
			END_IF;
			CustomVIndex := CustomVIndex + 1;
			IF CustomVTable[CustomVIndex] <= InvalidDistREAL THEN
				CustomVIndex := 1;
			END_IF;
			IF CustomVHits <= 0 THEN
				MakeCustomVTable := TRUE;
				CustomVIndex := 0;
			END_IF;
		END_IF;
		IF BeadRollUsedUp THEN
			IF BeadRollHits > 0 THEN
				BeadRollFires := TRUE;
				BeadRollHits := BeadRollHits - 1;
			END_IF;
			BeadRollIndex := BeadRollIndex + 1;
			IF BeadRollTable[BeadRollIndex] <= InvalidDistREAL THEN
				BeadRollIndex := 1;
			END_IF;
			IF BeadRollHits <= 0 THEN
				MakeBeadRollTable := TRUE;
				BeadRollIndex := 0;
			END_IF;
	    END_IF;
	END_IF;
END_ACTION
```
